// TwinCAT 3 PLC project PLC1
// ProgramVersion: 3.1.4024.12
// libraries:
//   Tc2_Standard, * (Beckhoff Automation GmbH)
//   Tc2_System, * (Beckhoff Automation GmbH)
//   Tc3_Module, * (Beckhoff Automation GmbH)
// project tree:
//   GVLs/ Grinder.TcGVL
//   / PlcTask.TcTTO
//   POUs/ MAIN.TcPOU, MAIN2.TcPOU, RunGrindingWheel.TcPOU
// real-time tasks:
//   TASK PlcTask: cycle T#1ms, priority 20, ADS port 350

CONFIGURATION PLC1
    RESOURCE PLC ON TwinCAT3
        TASK PlcTask(INTERVAL := T#1ms, PRIORITY := 20);
        PROGRAM MAIN WITH PlcTask : MAIN;
    END_RESOURCE
END_CONFIGURATION

// ---- GVLs/Grinder.TcGVL
{attribute 'qualified_only'}
VAR_GLOBAL
	GrindingWheelMS : BOOL;
	StartGrindingWheelPB : BOOL;
	StopGrindingWheelPB : BOOL;
END_VAR

// ---- POUs/MAIN.TcPOU
PROGRAM MAIN
VAR
END_VAR

RunGrindingWheel();

END_PROGRAM

// ---- POUs/RunGrindingWheel.TcPOU
PROGRAM RunGrindingWheel
VAR
END_VAR

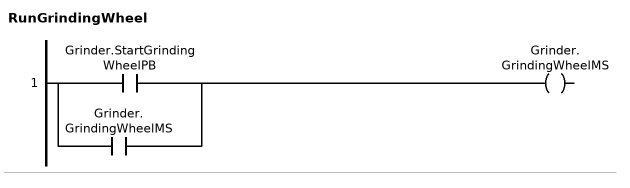
// NETWORK 1
Grinder.GrindingWheelMS := Grinder.StartGrindingWheelPB OR Grinder.GrindingWheelMS;

END_PROGRAM

// ---- POUs/MAIN2.TcPOU
PROGRAM MAIN2
VAR
	btn			:BOOL;
	btnStart	: BOOL;
	btnStop 	: BOOL := TRUE;
	Coil: BOOL;
	
END_VAR

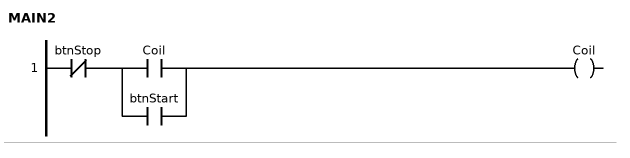
// NETWORK 1
Coil := NOT btnStop AND (Coil OR btnStart);

END_PROGRAM
